// TIA Portal project "Simple-Motor-Control" (V18)

(* hardware
DEVICE "S7-1500/ET200MP station_1"  S7-1500 station
   slot 0: "Rail_0"  Rack  6ES7 590-1***0-0AA0
   slot 1: "Brain"  CPU 1511C-1 PN  6ES7 511-1CK01-0AB0  V2.9
      slot 3: "CPU display_1"  6ES7591-1AA00-0AA0
      slot 32768: "PROFINET interface_1"  X1
         slot 32769: "Port_1"  X1 P1
         slot 32770: "Port_2"  X1 P2
      slot 34817: "Virtual CP interface port_1"  Virtual CP interface port  Virtual CP interface port
DEVICE "HMI_1"  TP700 Comfort
   slot 0: "HMI_1"  TP700 Comfort  6AV2 124-0GC01-0AX0  17.0.0.0
   slot 1: "HMI_RT_1"  TP700 Comfort  6AV2 124-0GC01-0AX0  17.0.0.0
   slot 5: "HMI_1.IE_CP_1"  PROFINET Interface  17.0.0.0
      slot 1: "PROFINET Interface_1"  PROFINET Interface
         slot 1: "Port_1"  Port
         slot 2: "Port_2"  Port
   slot 7: "HMI_1.MPI/DP_CP_1"  MPI/DP Interface  17.0.0.0
*)

// ===== PLC "Brain"  CPU 1511C-1 PN =====

VAR_GLOBAL   // PLC tag table "Default tag table"
   "iStart_PB" AT %M0.0 : Bool;   // Start Push Button Input
   "iStop_PB" AT %M0.1 : Bool;   // Stop Push Button Input (NC Logic)
   "iOverload_Fault" AT %I0.2 : Bool;   // Motor Thermal Overload Input
   "qMotor_On" AT %Q0.0 : Bool;   // Command to run the Motor
   "qFault_Status" AT %Q0.1 : Bool;   // Fault Indicator Status
END_VAR

ORGANIZATION_BLOCK "Main"   // OB1, LAD, ProgramCycle
TITLE = "Main Program Sweep (Cycle)"
{ S7_Optimized_Access := 'TRUE' }
VERSION : 0.1
   VAR_INPUT
      Initial_Call : Bool;   // Initial call of this OB
      Remanence : Bool;   // =True, if remanent data are available
   END_VAR
BEGIN

REGION Network 1: Command to run the Motor
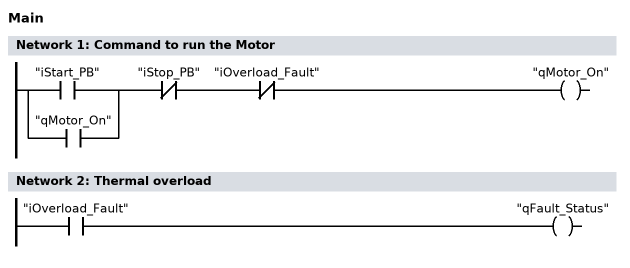
   RUNG wire#powerrail
      Contact( "iStart_PB" )
      wire#w1
      I_Contact( "iStop_PB" )
      I_Contact( "iOverload_Fault" )
      Coil( "qMotor_On" )
   END_RUNG
   RUNG wire#powerrail
      Contact( "qMotor_On" )
   END_RUNG wire#w1
   // the same network as SCL:
   "qMotor_On" := ("iStart_PB" OR "qMotor_On") AND NOT "iStop_PB" AND NOT "iOverload_Fault";
END_REGION

REGION Network 2: Thermal overload
   RUNG wire#powerrail
      Contact( "iOverload_Fault" )
      Coil( "qFault_Status" )
   END_RUNG
   // the same network as SCL:
   "qFault_Status" := "iOverload_Fault";
END_REGION
END_ORGANIZATION_BLOCK

(* ===== HMI "HMI_RT_1" =====
system functions are stored by id; their names below are inferred from use
connection "HMI_Connection_1": ETHERNET, S7_1500_OMS

HMI tags "Default tag table"
   "iOverload_Fault" : Bool = PLC iOverload_Fault AT %I0.2, 100 ms
   "iStart_PB" : Bool = PLC iStart_PB AT %M0.0, 100 ms
   "iStop_PB" : Bool = PLC iStop_PB AT %M0.1, 100 ms
   "qMotor_On" : Bool = PLC qMotor_On AT %Q0.0, 100 ms

screen "Root screen" 800x480, template "Template_1"
   Button "Button_1" at 36,30 size 123x70; TextOff 'Start'
      on Press: SetBit("iStart_PB")
      on Release: ResetBit("iStart_PB")
   Button "Button_2" at 608,364 size 119x73; TextOff 'Stop'
      on Press: SetBit("iStop_PB")
      on Release: ResetBit("iStop_PB")
   SymbolLibrary "Symbol library_1" at 0,184 size 386x223
      Appearance <- "qMotor_On"
   Circle "Circle_1" at 391,9 size 344x344
      Visibility <- "iOverload_Fault"
   TextField "Text field_1" at 344,142 size 423x99; Text 'Thermal Overload'
      Visibility <- "iOverload_Fault"
   TextField "Text field_3" at 10,232 size 423x99; Text 'Thermal Overload'
      Visibility <- "iOverload_Fault"
*)